Staubli VAL3: SpecialSeqVal.pjx

--- SpecialSeqVal.pjx ---
Parameters version=s7.8.1 stackSize=5000 millimeterUnit=true
Program file=start.pgx
Program file=stop.pgx
Data file=SpecialSeqVal.dtx

--- SpecialSeqVal.dtx ---
public num START_TRAJ_DOWN
public num START_TRAJ_STRE
public num END_TRAJECTORY
public num STOP_TRAJECTORY
